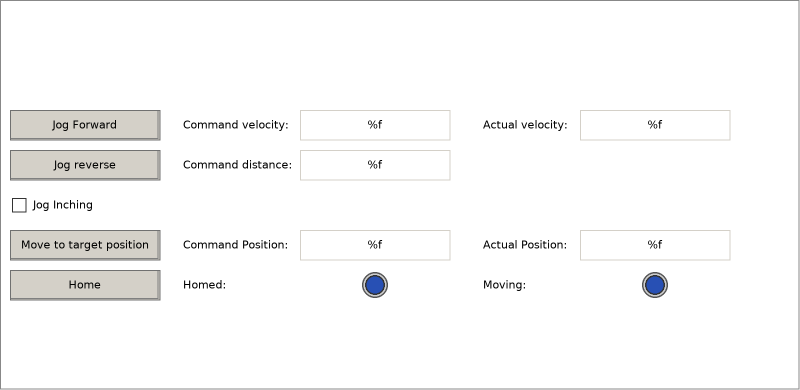
VISUALIZATION VisuAxisControl  // 800x390
VAR_IN_OUT
	pDev : POINTER TO Fb_DevAxis; 
END_VAR
    Button (10,110 150x30), "Jog Forward"
        tap pDev^.stManualCtrl.bCmdJogForward
    Button (10,150 150x30), "Jog reverse"
        tap pDev^.stManualCtrl.bCmdJogReverse
    Button (10,230 150x30), "Move to target position"
        tap pDev^.stManualCtrl.bCmdToPos
    Button (10,270 150x30), "Home"
        tap pDev^.stManualCtrl.bCmdHome
    Checkbox (10,190 150x30), "Jog Inching", variable: pDev^.stManualCtrl.bCmdInching
    Label (180,150 120x30), "Command distance:"
    Label (180,110 120x30), "Command velocity:"
    Label (180,230 120x30), "Command Position:"
    Textfield (300,110 150x30), "%f", text variable: pDev^.stManualCtrl.fVelocity
        OnMouseDown: write the text variable via VisuDialogs.Numpad
    Textfield (300,150 150x30), "%f", text variable: pDev^.stManualCtrl.fDistance
        OnMouseDown: write the text variable via VisuDialogs.Numpad
    Textfield (300,230 150x30), "%f", text variable: pDev^.stManualCtrl.fPosition
        OnMouseDown: write the text variable via VisuDialogs.Numpad
    Label (480,110 100x30), "Actual velocity:"
    Label (480,230 100x30), "Actual Position:"
    Textfield (580,230 150x30), "%f", text variable: pDev^.fActPosition
        OnMouseDown: write the text variable via VisuDialogs.Numpad
    Textfield (580,110 150x30), "%f", text variable: pDev^.fVelocity
        OnMouseDown: write the text variable via VisuDialogs.Numpad
    Lamp1 (580,270 150x30), variable: pDev^.AxisRef.Status.Moving, style: Lamp-Lamp1-Blue
    Label (480,270 100x30), "Moving:"
    Lamp1 (300,270 150x30), variable: pDev^.AxisRef.Status.Homed, style: Lamp-Lamp1-Blue
    Label (180,270 120x30), "Homed:"
END_VISUALIZATION

(* stored: Version 1.1.0.1, ProductVersion 3.1.4024.11
   Visu VisuAxisControl: Id {1ef75e37-be8d-09ba-01e3-08b392cb5229} *)
